RoboDK station: RS_dual_kuka_station_06_06.rdk

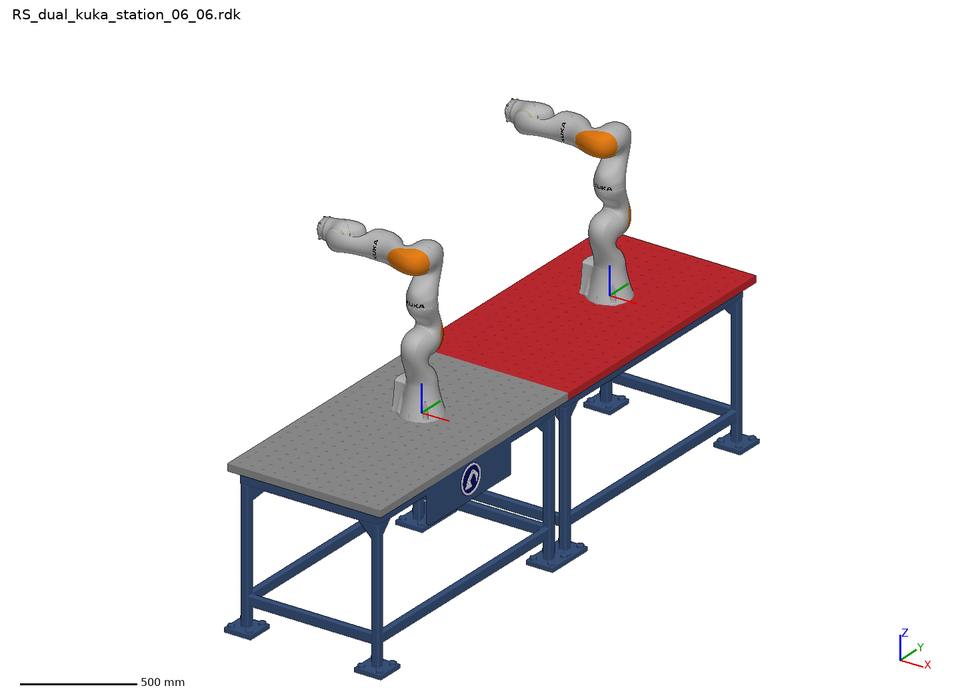
[picture v0: the station drawn from its stored meshes, robots at their saved joint values, targets as dots, program paths as lines]
Station dual_arm_station (saved by RoboDK 5.7.0). Poses are relative to the parent item; angles as X-Y-Z fixed-axis rotations.
Station parameters (name, value as stored): LIN64
  - Python program Prog1 (listed below)
  - object Table 1400x800x800mm at (0, -340, 0) mm, rotated rx 0 ry 0 rz -90 deg, size 1420 x 820 x 800 mm, geometry from Table-1400x800x800mm.sld
  - object Table 1400x800x800mm at (0, 340, 0) mm, rotated rx 0 ry 0 rz 90 deg, size 1420 x 820 x 800 mm, geometry from Table-1400x800x800mm.sld
  - frame robot0_base at (0, 880, 0) mm
    - robot robot0 (model KUKA LBR iiwa 7 R800): 7 axes, payload 7 kg, reach 800 mm, repeatability 0.1 mm, weight 23.9 kg
        modified DH rows (alpha deg, a mm, theta deg, d mm): 0, 0, 0, 340; -90, 0, 0, 0; 90, 0, 0, 400; -90, 0, 0, 0; 90, 0, 0, 400; -90, 0, 0, 0; 90, 0, 0, 130
        joint limits [-170, -120, -170, -120, -170, -120, -175] to [170, 120, 170, 120, 170, 120, 175]; home [0, 0, 0, -90, 0, 0, 0]; saved at [0, 0, 0, -90, 0, 0, 0]
      - tool Tool 1, TCP at (0, 0, 200) mm
  - frame robot1_base at (0, -520, 0) mm
    - robot robot1 (model KUKA LBR iiwa 7 R800): 7 axes, payload 7 kg, reach 800 mm, repeatability 0.1 mm, weight 23.9 kg
        modified DH rows (alpha deg, a mm, theta deg, d mm): 0, 0, 0, 340; -90, 0, 0, 0; 90, 0, 0, 400; -90, 0, 0, 0; 90, 0, 0, 400; -90, 0, 0, 0; 90, 0, 0, 130
        joint limits [-170, -120, -170, -120, -170, -120, -175] to [170, 120, 170, 120, 170, 120, 175]; home [0, 0, 0, -90, 0, 0, 0]; saved at [0, 0, 0, -90, 0, 0, 0]
      - tool Tool 2, TCP at (0, 0, 200) mm

--- Python program Prog1 ---
# Type help("robodk.robolink") or help("robodk.robomath") for more information
# Press F5 to run the script
# Documentation: https://robodk.com/doc/en/RoboDK-API.html
# Reference:     https://robodk.com/doc/en/PythonAPI/robodk.html
# Note: It is not required to keep a copy of this file, your Python script is saved with your RDK project

# You can also use the new version of the API:
from robodk import robolink    # RoboDK API
from robodk import robomath    # Robot toolbox
RDK = robolink.Robolink()

# Forward and backwards compatible use of the RoboDK API:
# Remove these 2 lines to follow python programming guidelines
from robodk import *      # RoboDK API
from robolink import *    # Robot toolbox
# Link to RoboDK
# RDK = Robolink()

# Notify user:
print('To edit this program:\nright click on the Python program, then, select "Edit Python script"')

# Program example:
item = RDK.Item('base')
if item.Valid():
    print('Item selected: ' + item.Name())
    print('Item posistion: ' + repr(item.Pose()))

print('Items in the station:')
itemlist = RDK.ItemList()
print(itemlist)

# Provoking an exception will display the console output if you run this script from RoboDK
raise Exception('Program not edited.')
